GLOBALCONSTANTS DefaultPool (* Global constants *)
  (* Standard: 61499-1 *)
  (* Version 1.0, 2024-02-25, franz *)
  VAR_GLOBAL CONSTANT
    ISO_DESIGNATOR_WIDTH : UINT := 80;
    ISO_DESIGNATOR_HEIGHT : UINT := 80;
    ISO_MASK_SIZE : UINT := 480;
    ISO_VERSION_LABEL : STRING := '       ';
    MASK_WIDTH : UINT := 480;
    MASK_HEIGHT : UINT := 480;
    WorkingSet_0 : UINT := 0;
    Macro_Go_To_DataMask_M1 : UINT := 1;
    Macro_Go_To_DataMask_M2 : UINT := 2;
    DataMask_M1 : UINT := 1000;
    DataMask_M2 : UINT := 1001;
    Container_B : UINT := 3000;
    SoftKeyMask_S1 : UINT := 4000;
    SoftKey_F1 : UINT := 5000;
    SoftKey_F2 : UINT := 5001;
    SoftKey_F3 : UINT := 5002;
    SoftKey_F4 : UINT := 5003;
    SoftKey_F5 : UINT := 5004;
    SoftKey_F6 : UINT := 5005;
    SoftKey_F7 : UINT := 5006;
    SoftKey_F8 : UINT := 5007;
    SoftKey_F9 : UINT := 5008;
    SoftKey_F10 : UINT := 5009;
    SoftKey_F11 : UINT := 5010;
    SoftKey_F12 : UINT := 5011;
    Button_A1 : UINT := 6000;
    Button_A2 : UINT := 6001;
    InputNumber_I1 : UINT := 9000;
    InputNumber_I2 : UINT := 9001;
    OutputString_WorkingSet_0 : UINT := 11000;
    OutputString_SoftKey_F1 : UINT := 11001;
    OutputString_SoftKey_F2 : UINT := 11002;
    OutputString_SoftKey_F3 : UINT := 11003;
    OutputString_SoftKey_F4 : UINT := 11004;
    OutputString_SoftKey_F5 : UINT := 11005;
    OutputString_SoftKey_F6 : UINT := 11006;
    OutputString_SoftKey_F7 : UINT := 11007;
    OutputString_SoftKey_F8 : UINT := 11008;
    OutputString_SoftKey_F9 : UINT := 11009;
    OutputString_SoftKey_F10 : UINT := 11010;
    OutputString_SoftKey_F11 : UINT := 11011;
    OutputString_SoftKey_F12 : UINT := 11012;
    OutputString_DataMask_M1 : UINT := 11013;
    OutputString_DataMask_M2 : UINT := 11014;
    OutputString_Go_To_DataMask_M1 : UINT := 11015;
    OutputString_Go_To_DataMask_M2 : UINT := 11016;
    OutputString_Button_A1 : UINT := 11017;
    OutputString_Button_A2 : UINT := 11018;
    OutputString_OutputNumber_N1 : UINT := 11019;
    OutputString_OutputNumber_N2 : UINT := 11020;
    OutputString_InputNumber_I1 : UINT := 11021;
    OutputNumber_N1 : UINT := 12000;
    OutputNumber_N2 : UINT := 12001;
    Line_W : UINT := 13000;
    Line_S : UINT := 13001;
    Logos_icon : UINT := 20000;
    FontAttributes_6x8 : UINT := 23000;
    FontAttributes_8x12 : UINT := 23001;
    FontAttributes_12x16 : UINT := 23002;
    FontAttributes_23003 : UINT := 23003;
    LineAttributes_black : UINT := 24000;
    ObjectPointer_P1 : UINT := 27000;
    AuxFunction2_X1 : UINT := 31000;
  END_VAR
END_GLOBALCONSTANTS
